// TIA Portal V17 export
// export: Created 2025-03-05T07:58:41.6276204Z, ExportSetting WithDefaults, DisplayName Totally Integrated Automation Portal, DisplayVersion V17 Update 8, DisplayName TIA Portal Openness, DisplayVersion V17 Update 8, DisplayName TIA Portal Version Control Interface, DisplayVersion V17, DisplayName SINAMICS Startdrive Advanced, DisplayVersion V17 SP2, DisplayName SINAMICS Startdrive G110M, G120, G120C, G120D, G120P, G115D, DisplayVersion V17 SP2, DisplayName SINAMICS Startdrive G130, G150, S120, S150, SINAMICS MV, S210, DisplayVersion V17 SP2, DisplayName STEP 7 Professional, DisplayVersion V17 Update 8, DisplayName SINUMERIK ONE STEP 7 Toolbox, DisplayVersion V17 Update 12, DisplayName SINUMERIK 840D sl STEP 7 Toolbox, DisplayVersion V17 Update 12, DisplayName STEP 7 Safety, DisplayVersion V17 Update 6, DisplayName WinCC Advanced, DisplayVersion V17 Update 8
DATA_BLOCK "LBP_Internal1"   // DB25000
TITLE = Internal DB for basic program / DB interno para el programa básico / Interner DB für Grundprogramm
{ S7_Optimized_Access := 'TRUE'; DB_Accessible_From_OPC_UA := 'FALSE' }
AUTHOR : SINUMERIK
FAMILY : SINUMERIK_ONE
VERSION : 6.15
// DB only for internal use in the basic program / DB solo para uso interno en el programa básico / DB nur zur internen Verwendung im Grundprogramm
// stored: AutoNumber true, DBAccessibleFromOPCUA false, DBAccessibleFromWebserver true, IsOnlyStoredInLoadMemory false, IsRetainMemResEnabled false, IsWriteProtectedInAS true, MemoryReserve 100
   VAR
      McpCommIniData : Array[0..32] of Struct
         mcpType : Byte;
         mcpName : String;
         cycleMCPSend : Time;
         minMCPSend : Time;
         clientSendTimeout : Time;
         mcpSendTimeout : Time;
         mcpSendWarning : Time;
         cycleClientSend : Time;
         handwheelOption : Bool;
         paramDataLength : UInt;
         paramData : Array[1..5] of Byte;
         paramDataDckLength : UInt;
         paramDataDck : Array[1..5] of Byte;
      END_STRUCT;
      McpCommDomain : String := 'local.';
      McpCommMcp1 : Struct
         useIpAddress : Bool;
         ipAddress : Array[1..4] of USInt;
      END_STRUCT;
      McpCommMcp2 : Struct
         useIpAddress : Bool;
         ipAddress : Array[1..4] of USInt;
      END_STRUCT;
      McpCommHt : Struct
         useIpAddress : Bool;
         ipAddress : Array[1..4] of USInt;
      END_STRUCT;
      McpCommDck1 : Struct
         useIpAddress : Bool;
         ipAddress : Array[1..4] of USInt;
      END_STRUCT;
      McpCommDck2 : Struct
         useIpAddress : Bool;
         ipAddress : Array[1..4] of USInt;
      END_STRUCT;
      McpCommIdent : Struct
         useIpAddress : Bool;
         ipAddress : Array[1..4] of USInt;
      END_STRUCT;
   END_VAR
BEGIN
   McpCommIniData[0].mcpType := 16#0080;
   McpCommIniData[1].mcpType := 16#0081;
   McpCommIniData[2].mcpType := 16#0082;
   McpCommIniData[3].mcpType := 16#0083;
   McpCommIniData[4].mcpType := 16#0084;
   McpCommIniData[5].mcpType := 16#0085;
   McpCommIniData[6].mcpType := 16#0086;
   McpCommIniData[7].mcpType := 16#0087;
   McpCommIniData[8].mcpType := 16#0088;
   McpCommIniData[9].mcpType := 16#0089;
   McpCommIniData[10].mcpType := 16#008A;
   McpCommIniData[11].mcpType := 16#008B;
   McpCommIniData[12].mcpType := 16#008C;
   McpCommIniData[13].mcpType := 16#008D;
   McpCommIniData[14].mcpType := 16#008E;
   McpCommIniData[16].mcpType := 16#0090;
   McpCommIniData[17].mcpType := 16#0091;
   McpCommIniData[32].mcpType := 16#00A0;
   McpCommIniData[0].mcpName := 'MCP_483C';
   McpCommIniData[1].mcpName := 'MCP_483';
   McpCommIniData[2].mcpName := 'MCP_310';
   McpCommIniData[3].mcpName := 'MCP_OEM';
   McpCommIniData[4].mcpName := 'MCP_DMG';
   McpCommIniData[5].mcpName := 'HT_8';
   McpCommIniData[6].mcpName := 'TCU_DT';
   McpCommIniData[7].mcpName := 'MCP_MPP';
   McpCommIniData[8].mcpName := 'HT_2';
   McpCommIniData[9].mcpName := 'OP_08T';
   McpCommIniData[10].mcpName := 'MCP 310C PN';
   McpCommIniData[11].mcpName := 'MCP INDEX OEM';
   McpCommIniData[12].mcpName := 'RCU/TCU30';
   McpCommIniData[13].mcpName := 'MCP Interface PN';
   McpCommIniData[14].mcpName := 'VDCK';
   McpCommIniData[16].mcpName := 'MCP_398C';
   McpCommIniData[17].mcpName := 'HT_10';
   McpCommIniData[32].mcpName := 'MODULAR_MCP';
   McpCommIniData[0..7].cycleMCPSend := T#200MS;
   McpCommIniData[8].cycleMCPSend := T#50MS;
   McpCommIniData[9..14].cycleMCPSend := T#200MS;
   McpCommIniData[16].cycleMCPSend := T#200MS;
   McpCommIniData[17].cycleMCPSend := T#30MS;
   McpCommIniData[32].cycleMCPSend := T#30ms;
   McpCommIniData[0..5].minMCPSend := T#20MS;
   McpCommIniData[6].minMCPSend := T#50MS;
   McpCommIniData[7..8].minMCPSend := T#20MS;
   McpCommIniData[9].minMCPSend := T#50MS;
   McpCommIniData[10..11].minMCPSend := T#20MS;
   McpCommIniData[12].minMCPSend := T#50MS;
   McpCommIniData[13..14].minMCPSend := T#20MS;
   McpCommIniData[16].minMCPSend := T#20MS;
   McpCommIniData[17].minMCPSend := T#10MS;
   McpCommIniData[32].minMCPSend := T#10ms;
   McpCommIniData[0..13].clientSendTimeout := T#1S_500MS;
   McpCommIniData[14].clientSendTimeout := T#1S_200MS;
   McpCommIniData[16].clientSendTimeout := T#1S_500MS;
   McpCommIniData[17].clientSendTimeout := T#200MS;
   McpCommIniData[32].clientSendTimeout := T#200ms;
   McpCommIniData[0..13].mcpSendTimeout := T#1S_500MS;
   McpCommIniData[14].mcpSendTimeout := T#1S_200MS;
   McpCommIniData[16].mcpSendTimeout := T#1S_500MS;
   McpCommIniData[17].mcpSendTimeout := T#500MS;
   McpCommIniData[32].mcpSendTimeout := T#500ms;
   McpCommIniData[0..7].mcpSendWarning := T#600MS;
   McpCommIniData[8].mcpSendWarning := T#150MS;
   McpCommIniData[9..14].mcpSendWarning := T#600MS;
   McpCommIniData[16].mcpSendWarning := T#600MS;
   McpCommIniData[17].mcpSendWarning := T#200MS;
   McpCommIniData[32].mcpSendWarning := T#200ms;
   McpCommIniData[0..4].cycleClientSend := T#50MS;
   McpCommIniData[5..6].cycleClientSend := T#200MS;
   McpCommIniData[7..11].cycleClientSend := T#50MS;
   McpCommIniData[12].cycleClientSend := T#200MS;
   McpCommIniData[13].cycleClientSend := T#50MS;
   McpCommIniData[14].cycleClientSend := T#200MS;
   McpCommIniData[16].cycleClientSend := T#50MS;
   McpCommIniData[17].cycleClientSend := T#100MS;
   McpCommIniData[32].cycleClientSend := T#100ms;
   McpCommIniData[8].handwheelOption := true;
   McpCommIniData[0..5].paramDataLength := 5;
   McpCommIniData[6].paramDataLength := 3;
   McpCommIniData[7..8].paramDataLength := 5;
   McpCommIniData[9].paramDataLength := 3;
   McpCommIniData[10..11].paramDataLength := 5;
   McpCommIniData[12].paramDataLength := 3;
   McpCommIniData[13].paramDataLength := 5;
   McpCommIniData[14].paramDataLength := 3;
   McpCommIniData[16..17].paramDataLength := 5;
   McpCommIniData[32].paramDataLength := 2;
   McpCommIniData[0].paramData[1] := 16#0080;
   McpCommIniData[0].paramData[2] := 16#00C0;
   McpCommIniData[0].paramData[3] := 16#0007;
   McpCommIniData[0].paramData[4] := 16#000D;
   McpCommIniData[0].paramData[5] := 16#0051;
   McpCommIniData[1].paramData[1] := 16#0081;
   McpCommIniData[1].paramData[2] := 16#00C0;
   McpCommIniData[1].paramData[3] := 16#0007;
   McpCommIniData[1].paramData[4] := 16#000D;
   McpCommIniData[1].paramData[5] := 16#0051;
   McpCommIniData[2].paramData[1] := 16#0082;
   McpCommIniData[2].paramData[2] := 16#00C0;
   McpCommIniData[2].paramData[3] := 16#0007;
   McpCommIniData[2].paramData[4] := 16#000D;
   McpCommIniData[2].paramData[5] := 16#0051;
   McpCommIniData[3].paramData[1] := 16#0083;
   McpCommIniData[3].paramData[2] := 16#00C0;
   McpCommIniData[3].paramData[3] := 16#0007;
   McpCommIniData[3].paramData[4] := 16#000D;
   McpCommIniData[3].paramData[5] := 16#0051;
   McpCommIniData[4].paramData[1] := 16#0084;
   McpCommIniData[4].paramData[2] := 16#00C0;
   McpCommIniData[4].paramData[3] := 16#0009;
   McpCommIniData[4].paramData[4] := 16#000D;
   McpCommIniData[4].paramData[5] := 16#0051;
   McpCommIniData[5].paramData[1] := 16#0085;
   McpCommIniData[5].paramData[2] := 16#00C0;
   McpCommIniData[5].paramData[3..4] := 16#0007;
   McpCommIniData[5].paramData[5] := 16#0050;
   McpCommIniData[6].paramData[1] := 16#0086;
   McpCommIniData[6].paramData[2] := 16#0040;
   McpCommIniData[6].paramData[3] := 16#0001;
   McpCommIniData[7].paramData[1] := 16#0087;
   McpCommIniData[7].paramData[2] := 16#00C0;
   McpCommIniData[7].paramData[3] := 16#0007;
   McpCommIniData[7].paramData[4] := 16#000D;
   McpCommIniData[7].paramData[5] := 16#0051;
   McpCommIniData[8].paramData[1] := 16#0088;
   McpCommIniData[8].paramData[2] := 16#00C0;
   McpCommIniData[8].paramData[3] := 16#0013;
   McpCommIniData[8].paramData[4] := 16#0005;
   McpCommIniData[8].paramData[5] := 16#0050;
   McpCommIniData[9].paramData[1] := 16#0089;
   McpCommIniData[9].paramData[2] := 16#0040;
   McpCommIniData[9].paramData[3] := 16#0001;
   McpCommIniData[10].paramData[1] := 16#008A;
   McpCommIniData[10].paramData[2] := 16#00C0;
   McpCommIniData[10].paramData[3] := 16#0007;
   McpCommIniData[10].paramData[4] := 16#000D;
   McpCommIniData[10].paramData[5] := 16#0051;
   McpCommIniData[11].paramData[1] := 16#008B;
   McpCommIniData[11].paramData[2] := 16#00C0;
   McpCommIniData[11].paramData[3] := 16#0007;
   McpCommIniData[11].paramData[4] := 16#000D;
   McpCommIniData[11].paramData[5] := 16#0051;
   McpCommIniData[12].paramData[1] := 16#008C;
   McpCommIniData[12].paramData[2] := 16#0040;
   McpCommIniData[12].paramData[3] := 16#0001;
   McpCommIniData[13].paramData[1] := 16#008D;
   McpCommIniData[13].paramData[2] := 16#00C0;
   McpCommIniData[13].paramData[3] := 16#0009;
   McpCommIniData[13].paramData[4] := 16#000D;
   McpCommIniData[13].paramData[5] := 16#0051;
   McpCommIniData[14].paramData[1] := 16#008E;
   McpCommIniData[14].paramData[2] := 16#0040;
   McpCommIniData[14].paramData[3] := 16#0001;
   McpCommIniData[16].paramData[1] := 16#0090;
   McpCommIniData[16].paramData[2] := 16#00C0;
   McpCommIniData[16].paramData[3] := 16#0007;
   McpCommIniData[16].paramData[4] := 16#000D;
   McpCommIniData[16].paramData[5] := 16#0051;
   McpCommIniData[17].paramData[1] := 16#0091;
   McpCommIniData[17].paramData[2] := 16#00C0;
   McpCommIniData[17].paramData[3..4] := 16#0007;
   McpCommIniData[17].paramData[5] := 16#0050;
   McpCommIniData[32].paramData[1] := 16#A0;
   McpCommIniData[32].paramData[2] := 16#FF;
   McpCommIniData[1..7].paramDataDckLength := 3;
   McpCommIniData[9].paramDataDckLength := 3;
   McpCommIniData[12].paramDataDckLength := 3;
   McpCommIniData[14].paramDataDckLength := 3;
   McpCommIniData[17].paramDataDckLength := 3;
   McpCommIniData[32].paramDataDckLength := 2;
   McpCommIniData[1].paramDataDck[1] := 16#0081;
   McpCommIniData[1].paramDataDck[2] := 16#0040;
   McpCommIniData[1].paramDataDck[3] := 16#0001;
   McpCommIniData[2].paramDataDck[1] := 16#0082;
   McpCommIniData[2].paramDataDck[2] := 16#0040;
   McpCommIniData[2].paramDataDck[3] := 16#0001;
   McpCommIniData[3].paramDataDck[1] := 16#0083;
   McpCommIniData[3].paramDataDck[2] := 16#0040;
   McpCommIniData[3].paramDataDck[3] := 16#0001;
   McpCommIniData[4].paramDataDck[1] := 16#0084;
   McpCommIniData[4].paramDataDck[2] := 16#0040;
   McpCommIniData[4].paramDataDck[3] := 16#0001;
   McpCommIniData[5].paramDataDck[1] := 16#0085;
   McpCommIniData[5].paramDataDck[2] := 16#0040;
   McpCommIniData[5].paramDataDck[3] := 16#0001;
   McpCommIniData[6].paramDataDck[1] := 16#0086;
   McpCommIniData[6].paramDataDck[2] := 16#0040;
   McpCommIniData[6].paramDataDck[3] := 16#0001;
   McpCommIniData[7].paramDataDck[1] := 16#0087;
   McpCommIniData[7].paramDataDck[2] := 16#0040;
   McpCommIniData[7].paramDataDck[3] := 16#0001;
   McpCommIniData[9].paramDataDck[1] := 16#0089;
   McpCommIniData[9].paramDataDck[2] := 16#0040;
   McpCommIniData[9].paramDataDck[3] := 16#0001;
   McpCommIniData[12].paramDataDck[1] := 16#008C;
   McpCommIniData[12].paramDataDck[2] := 16#0040;
   McpCommIniData[12].paramDataDck[3] := 16#0001;
   McpCommIniData[14].paramDataDck[1] := 16#008E;
   McpCommIniData[14].paramDataDck[2] := 16#0040;
   McpCommIniData[14].paramDataDck[3] := 16#0001;
   McpCommIniData[17].paramDataDck[1] := 16#0091;
   McpCommIniData[17].paramDataDck[2] := 16#0040;
   McpCommIniData[17].paramDataDck[3] := 16#0001;
   McpCommIniData[32].paramDataDck[1] := 16#A0;
   McpCommIniData[32].paramDataDck[2] := 16#FF;
END_DATA_BLOCK
